(* Schneider Machine Expert - Basic project resolucao, file version 2.7.0.0 *)
(* ProjectInformations: Name=Novo projeto *)

HARDWARE
  Cpu 0: TM221CE24R
  EthernetConfiguration: NetworkName=M221, IpAllocationMode=FixedAddress, IpAddress=0.0.0.0, SubnetMask=0.0.0.0
  SerialLineConfiguration: Baud=Baud19200, Parity=ParityEven, DataBits=DataBits8, StopBits=StopBits1, PhysicalMedium=PhysicalMediumRs485, TransmissionMode=TransmissionModeModbusRtu, SlaveId=1, Addressing=SlaveAddressing
  MastTask: UsePeriodScanMode=false, PeriodScan=100
  FastTask: Period=255
  CpuBehavior: StartingMode=StartAsPreviousState, AutoSaveRamOnEeprom=true, WatchdogPeriod=250

SYMBOLS  (address, symbol, comment, settings)
  %M0       SIG_IN_BOT_A
  %M1       SIG_AUX_PULS_A
  %M2       SIG_PULS_A
  %M5       SIG_MULT_5
  %M10      SIG_OUT_LED_A
  %C0       C_MULT_5  [Preset=4]
  %I0.0     IN_BOT_A
  %Q0.1     OUT_LED_A

POU Entradas
  (* SectionNumber=1 *)

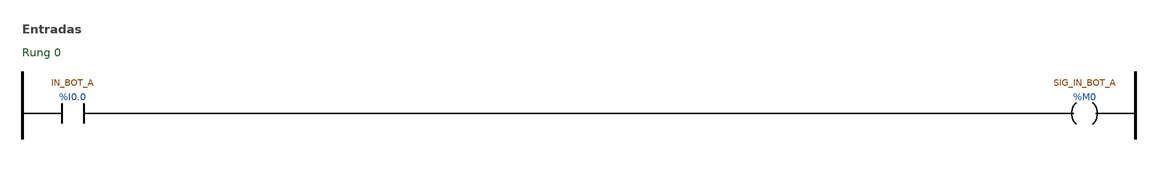

// Rung 0
  LD %I0.0                (* IN_BOT_A *)
  ST %M0                  (* SIG_IN_BOT_A *)
  // as ST:
  //   SIG_IN_BOT_A := IN_BOT_A;

POU Lógicas
  (* SectionNumber=2 *)

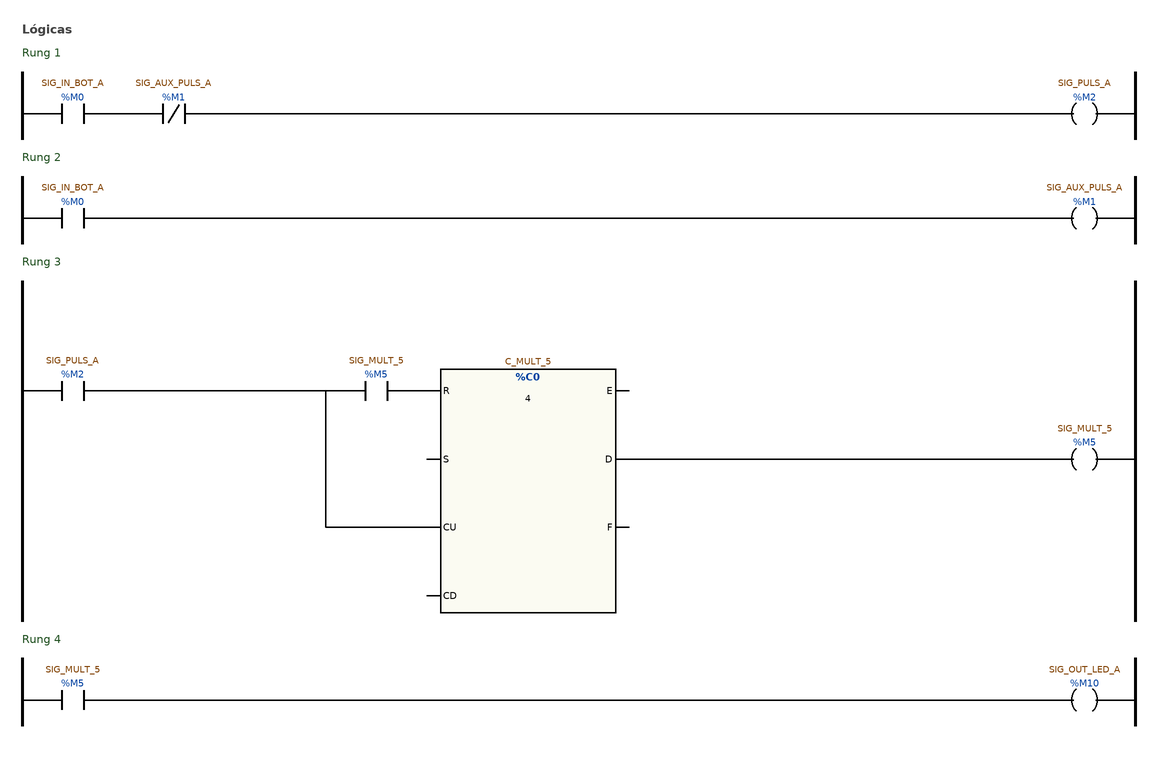

// Rung 1
  LD %M0                  (* SIG_IN_BOT_A *)
  ANDN %M1                (* SIG_AUX_PULS_A *)
  ST %M2                  (* SIG_PULS_A *)
  // as ST:
  //   SIG_PULS_A := SIG_IN_BOT_A AND NOT SIG_AUX_PULS_A;

// Rung 2
  LD %M0                  (* SIG_IN_BOT_A *)
  ST %M1                  (* SIG_AUX_PULS_A *)
  // as ST:
  //   SIG_AUX_PULS_A := SIG_IN_BOT_A;

// Rung 3
  BLK %C0                 (* C_MULT_5 *)
  LD %M2                  (* SIG_PULS_A *)
  MPS
  AND %M5                 (* SIG_MULT_5 *)
  R
  MPP
  CU
  OUT_BLK
  LD D
  ST %M5                  (* SIG_MULT_5 *)
  END_BLK
  // as ST:
  //   C_MULT_5(R := SIG_PULS_A AND SIG_MULT_5, CU := SIG_PULS_A);
  //   SIG_MULT_5 := C_MULT_5.D;

// Rung 4
  LD %M5                  (* SIG_MULT_5 *)
  ST %M10                 (* SIG_OUT_LED_A *)
  // as ST:
  //   SIG_OUT_LED_A := SIG_MULT_5;

POU Saídas
  (* SectionNumber=3 *)

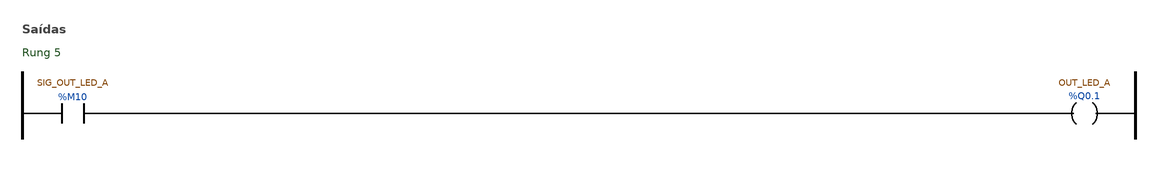

// Rung 5
  LD %M10                 (* SIG_OUT_LED_A *)
  ST %Q0.1                (* OUT_LED_A *)
  // as ST:
  //   OUT_LED_A := SIG_OUT_LED_A;
